Universal Robots PolyScope program: loop_91.urp

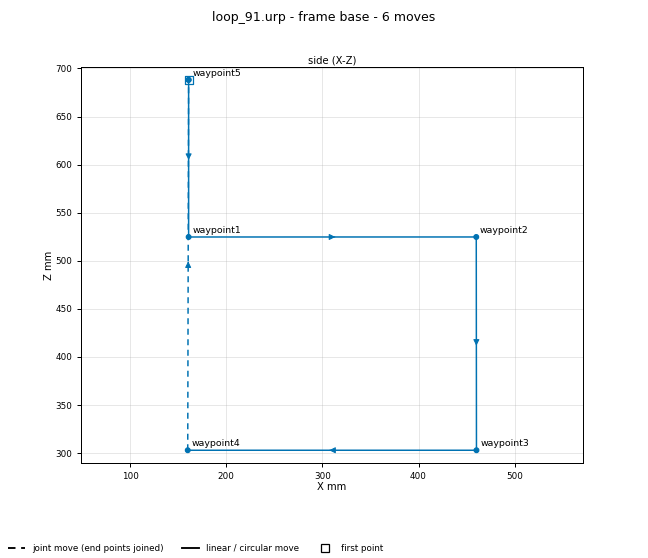
[picture p0: tool path of loop_91.urp in frame base, 6 of 6 moves have a stored position in this frame; points joined in program order, loops and branches not executed]
Program loop_91 (createdIn=3.2.19293 lastSavedIn=3.2.19293 directory=/programs installation=default robotSerialNumber=2015351391)
Calibrated DH parameters: a=[0.000352, -0.161198, -0.373486, 0.00005, 0.000049, 0]; d=[0.089268, 352.477598, -320.08558, -32.281492, 0.094939, 0.082518]; alpha=[1.570728, 0.001116, -0.003686, 1.571189, -1.570572, 0]; deltaTheta=[-0.000012, 1.181849, -1.491165, 0.309495, -0.000007, 0.000025]
Robot Program (runOnlyOnce=false motionType=MoveJ speed=1.047198 acceleration=1.396263 recalculateMotions=false)
  MoveJ speed 60 deg/s, acceleration 80 deg/s^2 (recalculateMotions=false)
    Waypoint waypoint5: TCP in base x=160.919 y=198.815 z=688.143 mm, rx=-1.5847 ry=-0.1115 rz=-0.2807 rad; joints [73.13, -59.949, -99.543, -21.223, 100.584, -14.682] deg
    Loop Counting (count=3) loopVariable(name=循环_1)
      MoveL speed 250 mm/s, acceleration 1200 mm/s^2 (recalculateMotions=false) feature=Base
        Waypoint waypoint1: TCP in base x=160.931 y=198.845 z=524.744 mm, rx=-1.5849 ry=-0.1114 rz=-0.2806 rad; joints [73.055, -56.065, -125.506, 0.863, 100.732, -14.67] deg
        Waypoint waypoint2: motionParameters(blendRadius=0.025); TCP in base x=460.019 y=198.808 z=524.767 mm, rx=-1.5849 ry=-0.1113 rz=-0.2806 rad; joints [28.366, -98.879, -92.608, 10.035, 145.495, -15.617] deg
        Waypoint waypoint3: TCP in base x=460.231 y=198.899 z=303.004 mm, rx=-1.5851 ry=-0.1093 rz=-0.2825 rad; joints [28.343, -113.123, -110.59, 42.388, 145.472, -15.457] deg
        Waypoint waypoint4: TCP in base x=160.006 y=198.932 z=303.001 mm, rx=-1.5851 ry=-0.1094 rz=-0.2825 rad; joints [73.337, -75.201, -152.72, 47.232, 100.456, -14.549] deg
  MoveJ speed 60 deg/s, acceleration 80 deg/s^2 (recalculateMotions=false)
    Waypoint waypoint5: TCP in base x=160.919 y=198.815 z=688.143 mm, rx=-1.5847 ry=-0.1115 rz=-0.2807 rad; joints [73.13, -59.949, -99.543, -21.223, 100.584, -14.682] deg
